// TIA Portal V20 export
ORGANIZATION_BLOCK "Interrupt1s"   // OB31, LAD, CyclicInterrupt
TITLE = Cyclic interrupt 100ms
AUTHOR : SICAR
FAMILY : OB
VERSION : 1.0
// organisation block
// stored: IsIECCheckEnabled true, SetENOAutomatically true
   VAR_INPUT
      Initial_Call : Bool;   // Initial call of this OB
      Event_Count : Int;   // Events discarded
   END_VAR
BEGIN

REGION Network 1: ChangeLog
   // Change log table:
   // Version | Date | Expert in charge | Changes applied
   // -------|---------|-------------|--------------------------------------------
   // 01.00.00 | 01.01.1999 | Person x | First released version
   // 01.00.01 | 02.01.1999 | Person y | Block was Updated
END_REGION

REGION Network 2: Call & measure-data into "EEmData_DB"
   // Call the energy efficiency monitor functions
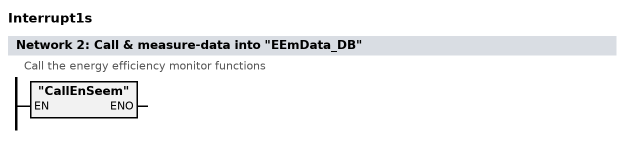
   RUNG wire#powerrail
      "CallEnSeem"()
   END_RUNG
   // the same network as SCL:
   "CallEnSeem"();
END_REGION
END_ORGANIZATION_BLOCK
